(* CODESYS project CmpTemplateTest.project

Project tree, tasks and I/O mapping:
  CODESYS_Control_Win : CODESYS Control Win V3, 3S - Smart Software Solutions GmbH, version 3.5.2.0
    application Application
      libraries: CmpTemplate, * (OEM)
      task T1 (cyclic, interval t#20ms, priority 1, watchdog t#50ms x 1) calls Main
      program Main [ST]
      function GenerateHardwareException [ST]
      function GenerateSoftwareException [ST]
      global variables GVL
  CODESYS_Control_Win_ExternalEvent : CODESYS Control Win V3 - External Event, 3S - Smart Software Solutions GmbH, version 3.5.4.0
    application Application
      libraries: CmpTemplate, * (OEM)
      task T1 (externalevent, external event MyEvent, priority 1, watchdog t#50ms x 1) calls Main
      program Main [ST]
  CODESYS_Control_Win_V3_64 : CODESYS Win Control for x64, 3S - Smart Software Solutions GmbH, version 3.5.6.0
    application Application
      libraries: CmpTemplate, * (OEM)
      task T1 (cyclic, interval t#20ms, priority 1, watchdog t#50ms x 1) calls Main
      global variables GVL
      function GenerateHardwareException [ST]
      function GenerateSoftwareException [ST]
      program Main [ST]
*)

// CODESYS_Control_Win_V3_64/Application/GVL
VAR_GLOBAL
	MyFB : MyExternalFunctionBlock;
END_VAR

// CODESYS_Control_Win/Application/GVL
VAR_GLOBAL
	MyFB : MyExternalFunctionBlock;
END_VAR

// CODESYS_Control_Win/Application/Main
PROGRAM Main
VAR
	xGenerateSoftwareException : BOOL;
	xGenerateHardwareException : BOOL;
	
	diFct : DINT;
	MyMessageText : STRING := 'Hello world!';
	dwTest : DWORD;
	dwSleepMs: DWORD := 1000;
	xTest : BOOL;
END_VAR

diFct := MyExternalFunction(diFct);
MyFB(MessageText := ADR(MyMessageText));
MyFB.PropTest := 123;
dwTest := MyFB.PropTest;
xTest := MyFB.MyMethod(10);

IF xGenerateSoftwareException THEN
	GenerateSoftwareException(dwSleepMs);
END_IF

IF xGenerateHardwareException THEN
	GenerateHardwareException();
END_IF

END_PROGRAM

// CODESYS_Control_Win_V3_64/Application/GenerateSoftwareException
FUNCTION GenerateSoftwareException : BOOL
VAR_INPUT
	dwSleepMs : DWORD;
END_VAR
VAR
END_VAR

MyFB.MySleep(dwSleepMs);

END_FUNCTION

// CODESYS_Control_Win/Application/GenerateSoftwareException
FUNCTION GenerateSoftwareException : BOOL
VAR_INPUT
	dwSleepMs : DWORD;
END_VAR
VAR
END_VAR

MyFB.MySleep(dwSleepMs);

END_FUNCTION

// CODESYS_Control_Win_V3_64/Application/GenerateHardwareException
FUNCTION GenerateHardwareException : BOOL
VAR_INPUT
END_VAR
VAR
END_VAR

MyFB.MyGenerateException(0);

END_FUNCTION

// CODESYS_Control_Win/Application/GenerateHardwareException
FUNCTION GenerateHardwareException : BOOL
VAR_INPUT
END_VAR
VAR
END_VAR

MyFB.MyGenerateException(0);

END_FUNCTION

// CODESYS_Control_Win_ExternalEvent/Application/Main
PROGRAM Main
VAR
	counter : DINT;
END_VAR

counter := counter + 1;

END_PROGRAM

// CODESYS_Control_Win_V3_64/Application/Main
PROGRAM Main
VAR
	xGenerateSoftwareException : BOOL;
	xGenerateHardwareException : BOOL;
	
	diFct : DINT;
	MyMessageText : STRING := 'Hello world!';
	dwTest : DWORD;
	dwSleepMs: DWORD := 1000;
	xTest : BOOL;
END_VAR

diFct := MyExternalFunction(diFct);
MyFB(MessageText := ADR(MyMessageText));
MyFB.PropTest := 123;
dwTest := MyFB.PropTest;
xTest := MyFB.MyMethod(10);

IF xGenerateSoftwareException THEN
	GenerateSoftwareException(dwSleepMs);
END_IF

IF xGenerateHardwareException THEN
	GenerateHardwareException();
END_IF

END_PROGRAM
